Universal Robots PolyScope program: Forces.urp

Program Forces (installation=default directory=/programs createdIn=5.9.3 lastSavedIn=5.14.5 robotSerialNumber=20195300809)
Calibrated DH parameters: a=[-0.000085, -0.20076, -0.212369, 0.000121, -0.000118, 0]; d=[0.15185, -26.306375, 24.753047, 1.684739, 0.085386, 0.092088]; alpha=[1.572149, -0.00522, -0.011864, 1.571339, -1.571085, 0]; deltaTheta=[0, 0.599885, -0.513355, -0.086555, 0.000006, 0]
InitVariablesNode
BeforeStart
  Script: socket_open("10.5.20.90",30002)
  str := "Start"
  Script: socket_send_string(str)
  miss := socket_read_string(timeout=3)
Robot Program (runOnlyOnce=false)
  MoveJ speed 5 deg/s, acceleration 80 deg/s^2 (useActiveTCP=true) feature=Base
    Waypoint Waypoint_1: TCP in base x=256.224 y=-262.417 z=131.748 mm, rx=0.8585 ry=3.0158 rz=0.0597 rad; joints [-26.889, -102.16, -68.275, -99.639, 91.579, 95.369] deg; TCP offset x=0 y=0 z=200 mm, rx=0 ry=0 rz=0 rad
    Waypoint Waypoint_2: TCP in base x=252.261 y=-265.907 z=155.628 mm, rx=0.856 ry=3.0141 rz=0.0317 rad; joints [-26.896, -102.534, -61.334, -105.866, 90.625, 95.366] deg
Thread Thread_1 (runOnlyOnce=false)
  Loop Forever
    Script: socket_open("10.5.20.90",30002)
    vector := get_tcp_force()
    fx := vector[0]
    fy := vector[1]
    fz := vector[2]
    mx := vector[3]
    my := vector[4]
    mz := vector[5]
    Script: socket_send_int(fx)
    Script: socket_send_int(fy)
    Script: socket_send_int(fz)
    Script: socket_send_int(mx)
    Script: socket_send_int(my)
    Script: socket_send_int(mz)
